//==================================================================================================
//								RJM Maszyny sp. z o.o.
//									13.05.2022
//
//	Obsługa przycisku niepodświetlanego
//	v1.0	|| TC v 3.1.4024.22		|| - pierwsza wersja
//==================================================================================================
FUNCTION_BLOCK FB_Przycisk_NO IMPLEMENTS I_Przycisk
VAR
	Wejscie							AT %I*	: BOOL;
END_VAR

//==================================================================================================
//								RJM Maszyny sp. z o.o.
//									13.05.2022
//
//	Sprawdzenie czy wciśnięty
//	v1.0	|| TC v 3.1.4024.22		|| - pierwsza wersja
//==================================================================================================
PROPERTY CzyNacisniety : BOOL
GET
CzyNacisniety								:= Wejscie;
END_GET
END_PROPERTY

//==================================================================================================
//								RJM Maszyny sp. z o.o.
//									13.05.2022
//
//	Sprawdzenie czy puszczony
//	v1.0	|| TC v 3.1.4024.22		|| - pierwsza wersja
//==================================================================================================
PROPERTY CzyPuszczony : BOOL
GET
CzyPuszczony								:= NOT Wejscie;
END_GET
END_PROPERTY

END_FUNCTION_BLOCK

(* stored: Version 1.1.0.1, ProductVersion 3.1.4024.11
   POU FB_Przycisk_NO: Id {67222b61-a5e6-41be-9a5c-281db6713395}, SpecialFunc None
   Property CzyNacisniety: Id {a51ec68c-ac56-4df6-bb60-e43aaa2ebf4e}
   Get Get: Id {028a46a3-9510-4918-9c72-1eba3fef1122}
   Property CzyPuszczony: Id {265ab40a-71ef-4ed7-aad2-b86894722f58}
   Get Get: Id {cb9ad17e-8555-45d9-8453-db0c589da2b4} *)
